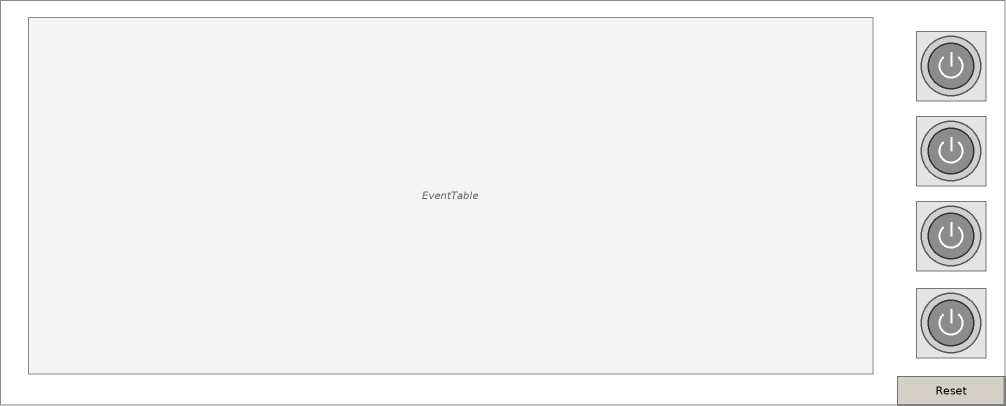
VISUALIZATION Visualization  // 1006x406
    EventTable (28,17 845x357)
        p1690906150: Class
        p3258520714: Date
        p2231227367: Time
        p3993844394: Time
        p2076579579: Details
        p3558512729: toHMI.aEvents
        p3921149237: m_pDataArray..pArray
    PowerSwitch (916,31 70x70), variable: prgAlarms.abAlarm[1], behaviour: TOGGLE, style: Switch-PowerSwitch-Gray
    PowerSwitch (916,116 70x70), variable: prgAlarms.abAlarm[2], behaviour: TOGGLE, style: Switch-PowerSwitch-Gray
    PowerSwitch (916,201 70x70), variable: prgAlarms.abAlarm[3], behaviour: TOGGLE, style: Switch-PowerSwitch-Gray
    PowerSwitch (916,288 70x70), variable: prgAlarms.abAlarm[4], behaviour: TOGGLE, style: Switch-PowerSwitch-Gray
    Button (897,376 109x30), "Reset"
        tap fromHMI.bIhmReset
END_VISUALIZATION

(* stored: Version 1.1.0.1, ProductVersion 3.1.4024.11
   Visu Visualization: Id {fc53fa3f-127d-4438-9ed7-9902ec9213d8} *)
